PROGRAM MAIN_ExternalTick_F
VAR
	state : INT := 0;	
	bStart : BOOL; 
	hint: STRING;
	hr: HRESULT;
	eCurrentMode: E_RtMode;
END_VAR

VAR_OUTPUT 
	value AT %Q* : UDINT;	
END_VAR

CASE state OF
	0:
		IF(bStart = TRUE) THEN 		
			state:= 1;
			value:=100; // steps to decrement as Cyclic
			hint := '..cycling...'; 		
		END_IF
	1:
		hr := F_UMRTGetTickMode(eCurrentMode);  
		IF(SUCCEEDED(hr) AND eCurrentMode = E_RtMode.RtMode_Cyclic) THEN 
			value:=value-1; //decrementing Cyclic (near realtime speed) 
			IF value = 0 THEN
				state := 2;
				value := 100; // Steps to decrement by External Ticks 
				hint := '!!! WAITING FOR EXTERNAL TICKS !!!'; 		
				F_UMRTChangeTickMode(E_RtMode.RtMode_Externaltick);
			END_IF
		ELSE 
			state := 97; 	
		END_IF
	2:
		hr := F_UMRTGetTickMode(eCurrentMode);  
		IF(SUCCEEDED(hr) AND eCurrentMode = E_RtMode.RtMode_Externaltick) THEN 
			value:=value-1; //decrementing as fast as possible 
			IF value = 0 THEN
				state := 0;
				hint := '..cycling (init)...'; 		
				(*switch back to cyclic mode*)		
				F_UMRTChangeTickMode(E_RtMode.RtMode_Cyclic);
			END_IF
		ELSE 
			state := 98; 	
		END_IF	
END_CASE

END_PROGRAM

(* stored: Version 1.1.0.1, ProductVersion 3.1.4025.18
   POU MAIN_ExternalTick_F: Id {b50c44e4-0af5-4535-a709-3ae5e67c7f1f}, SpecialFunc None *)
